PROGRAM main
VAR
	Q_READY AT %QX0.0 : bool := False;
	Q_REQUEST AT %QX0.1 : bool := False;
	Q_PASS_ALLOWED AT %QX0.2 : bool := False;
	Q_EMERGENCY AT %QX0.3 : bool := False;
	CMD_ROBOT_REQUEST AT %QX1.0 : bool := False;
	CMD_HMI_ALLOW AT %QX1.1 : bool := False;
	CMD_ROBOT_PASSED AT %QX1.2 : bool := False;
	CMD_EMERGENCY AT %QX1.3 : bool := False;
	CMD_RESET AT %QX1.4 : bool := False;
	STATUS_READY AT %QX0.4 : bool := False;
	STATUS_REQUEST AT %QX0.5 : bool := False;
	STATUS_PASS_ALLOWED AT %QX0.6 : bool := False;
	STATUS_EMERGENCY AT %QX0.7 : bool := False;
	STATUS_BARRIER_OPEN : bool := False;
	STATUS_PASS_PERMISSION : bool := False;
	M_READY : bool := True;
	M_REQUEST : bool := False;
	M_PASS_ALLOWED : bool := False;
	M_EMERGENCY : bool := False;
	PWM_CONTROLLER0 : PWM_CONTROLLER;
	SERVO_CHANNEL : sint := 13;
	SERVO_FREQ : real := 50.0;
	SERVO_DUTY_CLOSED : real := 5.0;
	SERVO_DUTY_OPEN : real := 7.5;
	PWM_CLOSE_OK : bool := False;
	PWM_OPEN_OK : bool := False;
	PWM_CONTROLLER1 : PWM_CONTROLLER;
	PWM_CONTROLLER2 : PWM_CONTROLLER;
END_VAR

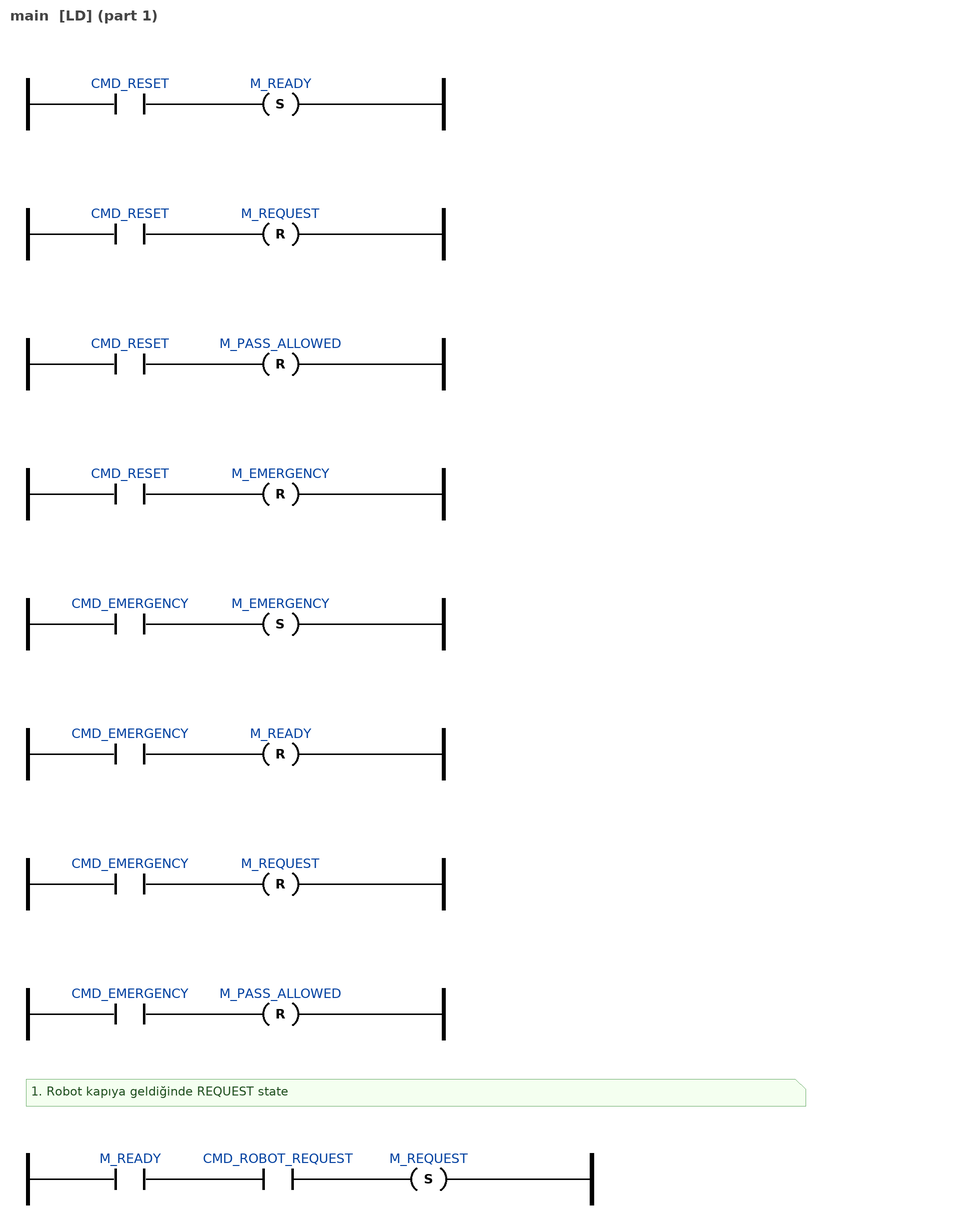
(* LD diagram, written out as Structured Text *)
IF CMD_RESET THEN M_READY := TRUE; END_IF;
IF CMD_RESET THEN M_REQUEST := FALSE; END_IF;
IF CMD_RESET THEN M_PASS_ALLOWED := FALSE; END_IF;
IF CMD_RESET THEN M_EMERGENCY := FALSE; END_IF;
IF CMD_EMERGENCY THEN M_EMERGENCY := TRUE; END_IF;
IF CMD_EMERGENCY THEN M_READY := FALSE; END_IF;
IF CMD_EMERGENCY THEN M_REQUEST := FALSE; END_IF;
IF CMD_EMERGENCY THEN M_PASS_ALLOWED := FALSE; END_IF;
(* 1. Robot kapıya geldiğinde REQUEST state *)
IF M_READY AND CMD_ROBOT_REQUEST THEN M_REQUEST := TRUE; END_IF;
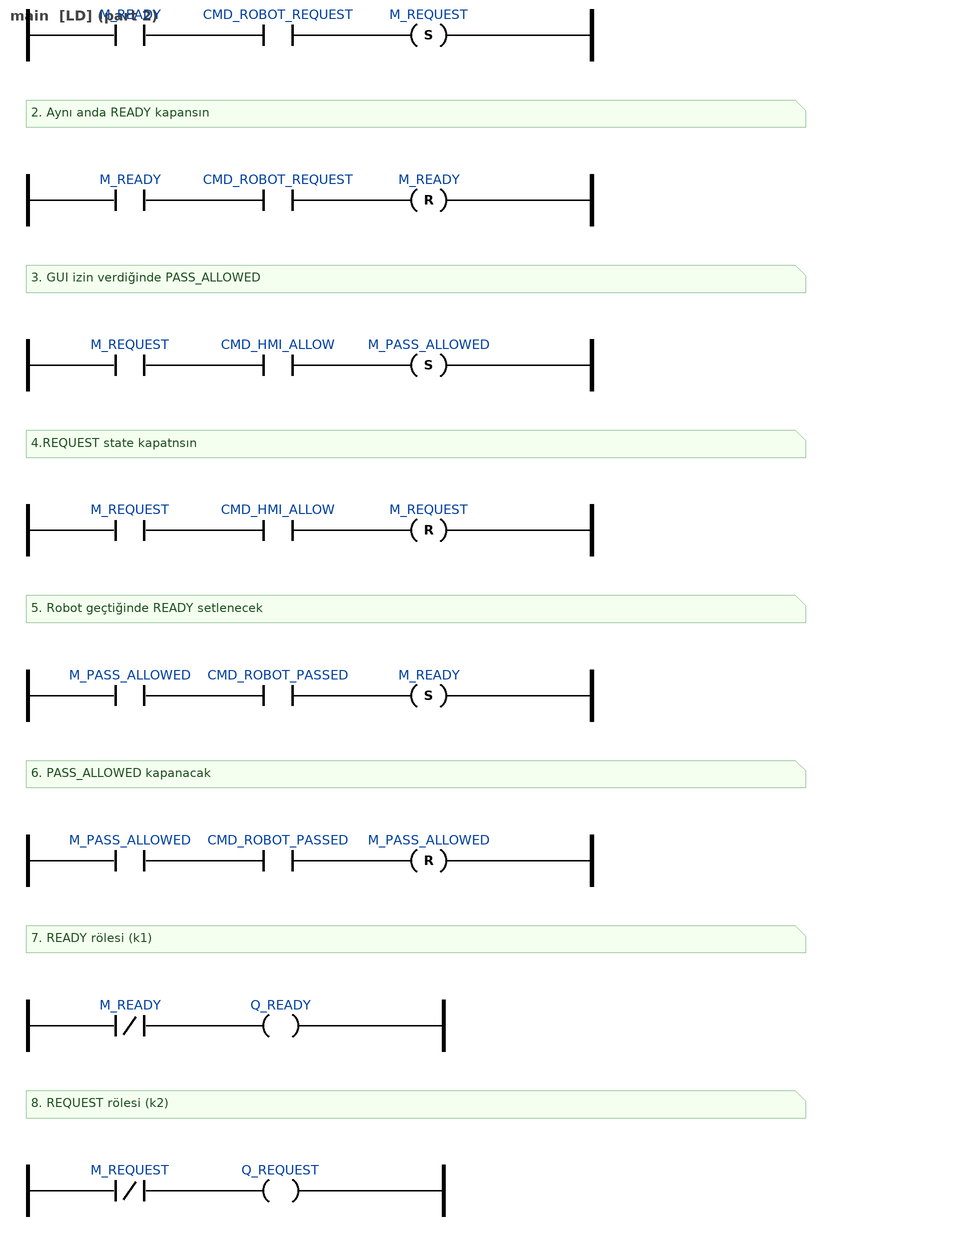
(* 2. Aynı anda READY kapansın *)
IF M_READY AND CMD_ROBOT_REQUEST THEN M_READY := FALSE; END_IF;
(* 3. GUI izin verdiğinde PASS_ALLOWED *)
IF M_REQUEST AND CMD_HMI_ALLOW THEN M_PASS_ALLOWED := TRUE; END_IF;
(* 4.REQUEST state kapatnsın *)
IF M_REQUEST AND CMD_HMI_ALLOW THEN M_REQUEST := FALSE; END_IF;
(* 5. Robot geçtiğinde READY setlenecek *)
IF M_PASS_ALLOWED AND CMD_ROBOT_PASSED THEN M_READY := TRUE; END_IF;
(* 6. PASS_ALLOWED kapanacak *)
IF M_PASS_ALLOWED AND CMD_ROBOT_PASSED THEN M_PASS_ALLOWED := FALSE; END_IF;
(* 7. READY rölesi (k1) *)
Q_READY := NOT M_READY;
(* 8. REQUEST rölesi (k2) *)
Q_REQUEST := NOT M_REQUEST;
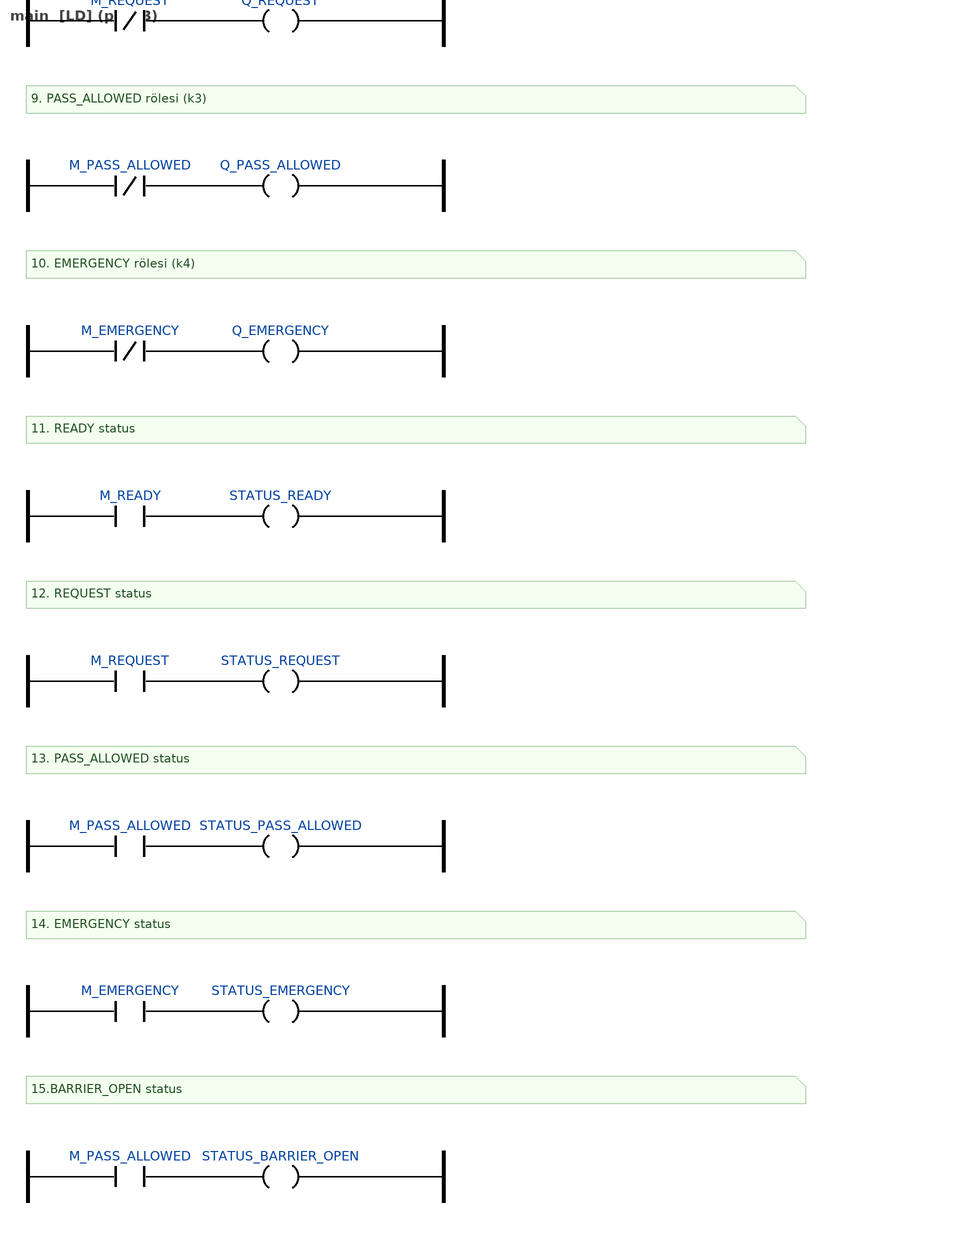
(* 9. PASS_ALLOWED rölesi (k3) *)
Q_PASS_ALLOWED := NOT M_PASS_ALLOWED;
(* 10. EMERGENCY rölesi (k4) *)
Q_EMERGENCY := NOT M_EMERGENCY;
(* 11. READY status *)
STATUS_READY := M_READY;
(* 12. REQUEST status *)
STATUS_REQUEST := M_REQUEST;
(* 13. PASS_ALLOWED status *)
STATUS_PASS_ALLOWED := M_PASS_ALLOWED;
(* 14. EMERGENCY status *)
STATUS_EMERGENCY := M_EMERGENCY;
(* 15.BARRIER_OPEN status *)
STATUS_BARRIER_OPEN := M_PASS_ALLOWED;
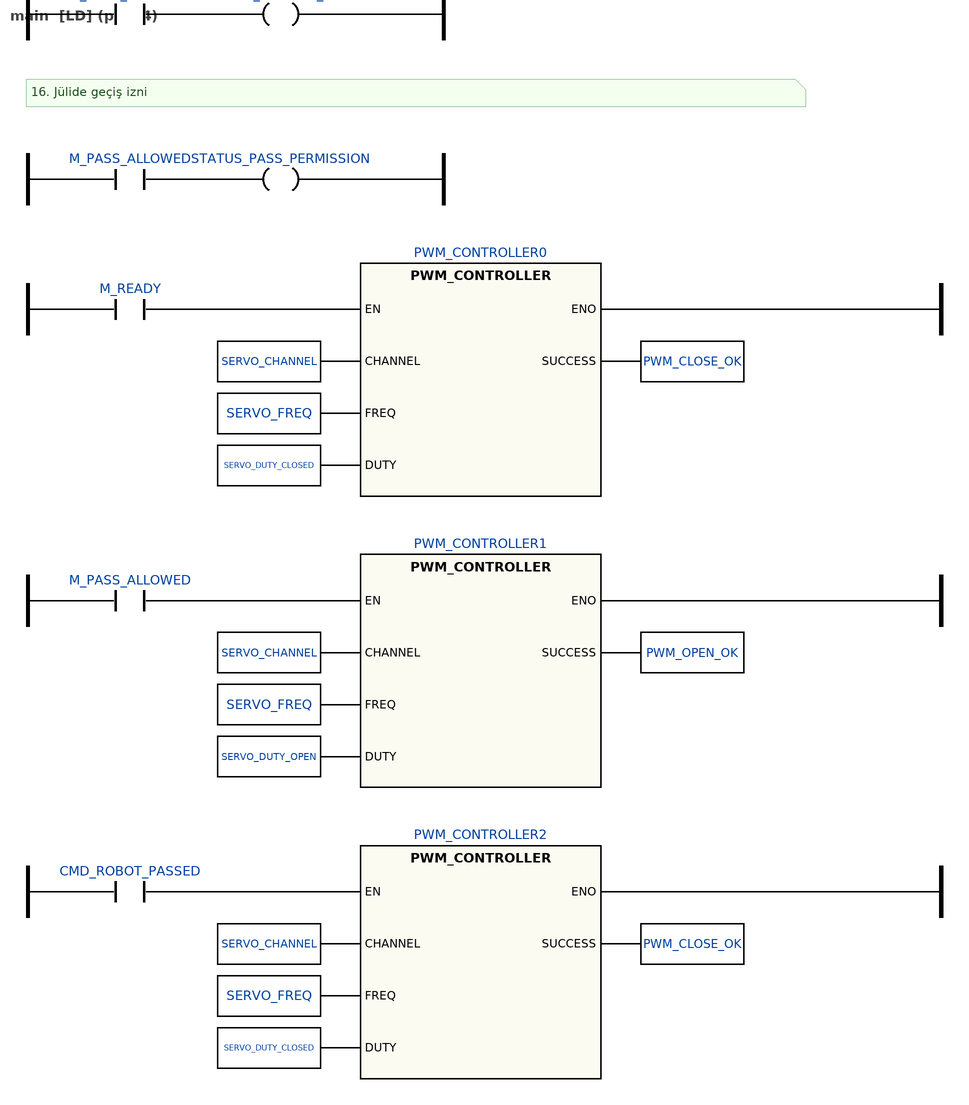
(* 16. Jülide geçiş izni *)
STATUS_PASS_PERMISSION := M_PASS_ALLOWED;
PWM_CONTROLLER0(EN := M_READY, CHANNEL := SERVO_CHANNEL, FREQ := SERVO_FREQ, DUTY := SERVO_DUTY_CLOSED);
IF PWM_CONTROLLER0.ENO THEN PWM_CLOSE_OK := PWM_CONTROLLER0.SUCCESS; END_IF;
PWM_CONTROLLER1(EN := M_PASS_ALLOWED, CHANNEL := SERVO_CHANNEL, FREQ := SERVO_FREQ, DUTY := SERVO_DUTY_OPEN);
IF PWM_CONTROLLER1.ENO THEN PWM_OPEN_OK := PWM_CONTROLLER1.SUCCESS; END_IF;
PWM_CONTROLLER2(EN := CMD_ROBOT_PASSED, CHANNEL := SERVO_CHANNEL, FREQ := SERVO_FREQ, DUTY := SERVO_DUTY_CLOSED);
IF PWM_CONTROLLER2.ENO THEN PWM_CLOSE_OK := PWM_CONTROLLER2.SUCCESS; END_IF;
END_PROGRAM
